FUNCTION_BLOCK E_F_TRIG (* Boolean falling edge detection *)
  (* Standard: 61499-1 Annex A; Description: Copyright (c) 2017 fortiss GmbH This program and the accompanying materials are made available under the terms of the Eclipse Public License 2.0 which is available at https://www.eclipse.org/legal/epl-2.0/ SPDX-License-Identifier: EPL-2.0 *)
  (* Version 1.0, 2017-09-22, Alois Zoitl, fortiss GmbH, initial API and implementation and/or initial documentation *)
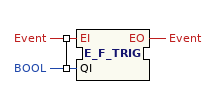
  EVENT_INPUT
    EI WITH QI; (* check for falling edge *)
  END_EVENT
  EVENT_OUTPUT
    EO; (* confirmation that an falling edge was detected *)
  END_EVENT
  VAR_INPUT
    QI : BOOL; (* value to check for a falling edge *)
  END_VAR
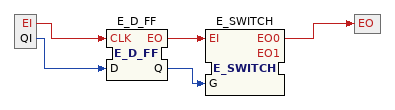
  FBS
    E_D_FF : E_D_FF;
    E_SWITCH : E_SWITCH;
  END_FBS
  EVENT_CONNECTIONS
    EI TO E_D_FF.CLK;
    E_D_FF.EO TO E_SWITCH.EI;
    E_SWITCH.EO0 TO EO;
  END_CONNECTIONS
  DATA_CONNECTIONS
    QI TO E_D_FF.D;
    E_D_FF.Q TO E_SWITCH.G;
  END_CONNECTIONS
END_FUNCTION_BLOCK
